Fanuc KAREL source: V_ADJ_2D.kl

PROGRAM T
%NOLOCKGROUP
VAR
 v0 : INTEGER
 v1 : REAL
 v2 : REAL
 v3 : INTEGER
BEGIN
 V_ADJ_2D(v0, v1, v2, v3)
END T
